FUNCTION Convert_UDINT_TO_DINT : BOOL
VAR_INPUT
	in : UDINT;
	out : REFERENCE TO DINT;
END_VAR
VAR
	converted : DINT;
END_VAR

converted := UDINT_TO_DINT(in);

IF (DINT_TO_UDINT(converted) <> in) THEN
	RETURN;
END_IF

out := converted;
Convert_UDINT_TO_DINT := TRUE;

END_FUNCTION

(* stored: Version 1.1.0.1, ProductVersion 3.1.4024.12
   POU Convert_UDINT_TO_DINT: Id {7d1801ea-3043-49ca-aeac-00449dddb2d8}, SpecialFunc None *)
